TEXTLIST WorkAreaLGVReq
  0 = 'Nop'
  1 = 'LGV Request'
  2 = 'LGV Ok In'
   = ''
END_TEXTLIST

(* stored: Version 1.1.0.1, ProductVersion 3.1.4024.11
   TextList WorkAreaLGVReq: Id {f2f13db0-fcaf-4a25-85fe-91c154214ddd} *)
